{attribute 'qualified_only'}
{attribute 'strict'}
TYPE
	E_Mode :
	(
		Auto := 0,
		Manual
	);
END_TYPE

(* stored: Version 1.1.0.1, ProductVersion 3.1.4024.12
   DUT E_Mode: Id {3aa44668-f60e-4867-abeb-842125046b29} *)
